PROGRAM StructureTesting
VAR
	aSensors : ARRAY[1..2] OF ST_Sensor;
END_VAR

//aSensors[1].scaledTemp := (aSensors[1].rawTemp)/327.67;
//aSensors[2].scaledTemp := (aSensors[2].rawTemp)/

aSensors[1].scaledTemp := F_Scaling(rawInput:= aSensors[1].rawTemp );

END_PROGRAM

(* stored: Version 1.1.0.1, ProductVersion 3.1.4024.12
   POU StructureTesting: Id {eecc1e57-15ee-49ce-a821-140cee8fcfdc}, SpecialFunc None *)
